// SIMATIC S7-200 project (STEP 7-Micro/WIN), CPU 221 REL 01.10

SYMBOL_TABLE USS Protocol
USS_LOW_V        VD1000   // (DWORD) Enter the starting address for USS Protocol symbols here.
USS_HIGH_V       VD1004
USS_TIME_OUT     VW1008
USS_I_LINE       VW1010
USS_DAT_PTR0     VD1012
USS_ACT_DRV0     VD1016
USS_CUR_DRV0     VD1020
USS_P0           V1024.0
USS_REQ_SNT0     V1024.1
USS_RETRY_P0     VB1025
USS_ERR_CODE     VB1026
USS_CS_D0        VD1027
USS_CS_W0        VW1027
USS_CS_W2        VW1029
USS_CS_B0        VB1027
USS_CS_B1        VB1028
USS_POLL_BUF     VB1031
USS_XMT_0        VB1046
USS_XMT_ADR0     VB1049
USS_X_STWD       VD1056
USS_X_BCC        VB1060
USS_X_DW1        VD1047
USS_X_DW5        VD1051
USS_X_DW9        VD1055
USS_X_DB13       VB1059
USS_RCV_BUF0     VB1061
USS_R_STX        VB1062
USS_R_LGE        VB1063
USS_R_ADR        VB1064
USS_R_STWD       VD1071
USS_R_DW1        VD1062
USS_R_DW5        VD1066
USS_R_DW9        VD1070
USS_R_W13        VW1074
USS_STAT_TAB     VB1076
USS_ADR_P0       VB1396
END_SYMBOL_TABLE

ORGANIZATION_BLOCK MAIN:OB1
TITLE=给某个德国制药厂定制的PLC程序。系统通过启动按钮启动，停止按钮停止。启动自锁标志只有在启动按钮按下或已置位，且停止按钮未按下时才能置位，确保系统在启动后持续运行直到操作员主动停止。启动后，循环计时器在启动自锁标志置位且计时器完成标志未置位时启动，计时10个时间单位，用于控制每个循环的时长。接着，循环计数器在循环计时器到时且计数器复位标志置位时递增，记录循环次数，预设值为60次。当循环计数器达到60时，计数器复位标志置位；此外，计时器完成标志在启动自锁标志置位且循环计时器到时置位，以协调计时和计数。在每个循环中，当循环计数器在0到53之间时，喷雾控制和风门控制在启动自锁标志置位且停止按钮未按下时激活，向物料喷洒液体并调节空气流通，实现湿化过程。而当循环计数器达到53到60之间时，摇振启动标志在启动自锁标志置位且停止按钮未按下时置位，同时关闭喷雾控制和风门控制，开始摇振操作。摇振过程通过摇振电磁阀控制实现，其在摇振启动标志置位且摇振通电计时器未到时激活。摇振通电计时器在摇振启动标志置位且摇振失电计时器未到时启动，计时10个时间单位；而后，摇振失电计时器在摇振通电计时器到时启动，计时10个时间单位。通过摇振通电计时器和摇振失电计时器的交替控制，摇振电磁阀控制实现周期性动作，驱动摇振机完成物料混合。为确保安全和正确运行，应在循环计数器超过60或启动自锁标志复位时复位摇振启动标志，以停止摇振操作，避免设备持续运行带来的潜在损坏或安全隐患。
BEGIN
Network 1 // 启动自锁
//  
// NETWORK COMMENTS
//  
// 
LD     I0.0
O      M0.2
AN     I1.0
=      M0.2
Network 2 // 计时基数设定
// 
// 
LD     M0.2
AN     M0.1
TON    T60, +10
Network 3 // 计数次数设置
// 
// 
LD     T60
LD     M0.0
CTU    C1, +60
Network 4 // 计数复位
// 
// 
LD     C1
=      M0.0
Network 5 // 喷雾和风门运行时间，同时使摇振复位
// 
// 
LD     M0.2
AN     I1.0
AW>=   C1, +0
AW<=   C1, +53
=      Q1.0
=      Q1.1
R      M0.3, 1
Network 6 // 复位喷雾/关排风阀门并开始启动摇振
// 
// 
LD     M0.2
AN     I1.0
AW>=   C1, +53
AW<=   C1, +60
=      M0.3
=      Q1.0
=      Q1.1
Network 7 // 复位T60 
// 
// 
LD     M0.2
A      T60
=      M0.1
Network 8 // 摇振电磁阀通电1S
// 
// 
LD     M0.3
AN     T46
TON    T45, +10
Network 9 // 摇振电磁阀失电1S
// 
// 
LD     T45
TON    T46, +10
Network 10 // 摇振标志Q0.0
// 
// 
LD     M0.3
AN     T45
=      Q0.0
END_ORGANIZATION_BLOCK
